TYPE ST_InfluxBuffer :
STRUCT
	Initialized : BOOL;
	ReadyToSend	: BOOL;
	Data 		: FB_STRINGBUILDER; 
END_STRUCT
END_TYPE

(* stored: Version 1.1.0.1, ProductVersion 3.1.4022.11
   DUT ST_InfluxBuffer: Id {5a54b913-84fc-42cd-8b14-4780d0b91fbc} *)
